# EPICS substitutions: db/Beckhoff_5XXX/ecmcEL5112_AB.substitutions
file "ecmcEL5131-chX.template"
{
    pattern {CH_ID}
            {01   }
            {02   }
}
